// TIA Portal V20 export
TYPE "UDT_ModeSt"
   STRUCT
      Bit0 : Bool;   // 0=Low Limit, 1=High Limit
      Bit1 : Bool;   // 1=Status Limit (purple)
      Bit2 : Bool;   // 1=Alarm Limit (red)
      Bit3 : Bool;   // 1=Warning Limit (yellow)
      Bit4 : Bool;   // Reserved
      Bit5 : Bool;   // Reserved
      Bit6 : Bool;   // Reserved
      Bit7 : Bool;   // Reserved
   END_STRUCT;
END_TYPE
